// TIA Portal V20 export
TYPE "typeCmControlNodeBrakeTest"
// stored: Namespace Unit1.Em2
   STRUCT
      jrOutPnPLeftAxisZ : "LER_typeBrakeTestEmControlNodes";
      jrOutPnPRightAxisZ : "LER_typeBrakeTestEmControlNodes";
   END_STRUCT;
END_TYPE
